(* IEC 61131-3 sources: com.logicals.lc3.webinar/usRTS_RPMControl_iSOC/src_FB_LIB_SAFE/Convert/ULINT, 4 files *)

(* ---- wTRUNC_ULINT_TO_UDINT.iecst ---- *)
NAMESPACE logicals.web.standard
NAMESPACE convert

/*
 * Function block wrapper for IEC 61131-3 TO_UDINT<br>
 * IN =  input value (ULINT)<br>
 * OUT = IN (UDINT)<br>
 */
FUNCTION_BLOCK wTRUNC_ULINT_TO_UDINT
	{ vNameAlignment:="center"; altName:="TRUNC_ULINT_TO_UDINT"; bgColor:="Plum"; width:=180; hideIONames; }
	VAR_INPUT
		IN : ULINT;
	END_VAR
	VAR_OUTPUT
		OUT: UDINT;
	END_VAR

	OUT := TO_UDINT(IN:=IN, ENO=>ENO);
END_FUNCTION_BLOCK

END_NAMESPACE
END_NAMESPACE

(* ---- wTRUNC_ULINT_TO_UINT.iecst ---- *)
NAMESPACE logicals.web.standard
NAMESPACE convert

/*
 * Function block wrapper for IEC 61131-3 TO_UINT<br>
 * IN =  input value (ULINT)<br>
 * OUT = IN (UINT)<br>
 */
FUNCTION_BLOCK wTRUNC_ULINT_TO_UINT
	{ vNameAlignment:="center"; altName:="TRUNC_ULINT_TO_UINT"; bgColor:="Plum"; width:=180; hideIONames; }
	VAR_INPUT
		IN : ULINT;
	END_VAR
	VAR_OUTPUT
		OUT: UINT;
	END_VAR

	OUT := TO_UINT(IN:=IN, ENO=>ENO);
END_FUNCTION_BLOCK

END_NAMESPACE
END_NAMESPACE

(* ---- wTRUNC_ULINT_TO_USINT.iecst ---- *)
NAMESPACE logicals.web.standard
NAMESPACE convert

/*
 * Function block wrapper for IEC 61131-3 TO_USINT<br>
 * IN =  input value (ULINT)<br>
 * OUT = IN (USINT)<br>
 */
FUNCTION_BLOCK wTRUNC_ULINT_TO_USINT
	{ vNameAlignment:="center"; altName:="TRUNC_ULINT_TO_USINT"; bgColor:="Plum"; width:=180; hideIONames; }
	VAR_INPUT
		IN : ULINT;
	END_VAR
	VAR_OUTPUT
		OUT: USINT;
	END_VAR

	OUT := TO_USINT(IN:=IN, ENO=>ENO);
END_FUNCTION_BLOCK

END_NAMESPACE
END_NAMESPACE

(* ---- wULINT_TO_LWORD.iecst ---- *)
NAMESPACE logicals.web.standard
NAMESPACE convert

/*
 * Function block wrapper for IEC 61131-3 TO_LWORD<br>
 * IN =  input value (ULINT)<br>
 * OUT = IN (LWORD)<br>
 */
FUNCTION_BLOCK wULINT_TO_LWORD
	{ vNameAlignment:="center"; altName:="ULINT_TO_LWORD"; bgColor:="DodgerBlue"; width:=140; hideIONames; }
	VAR_INPUT
		IN : ULINT;
	END_VAR
	VAR_OUTPUT
		OUT: LWORD;
	END_VAR

	OUT := TO_LWORD(IN:=IN, ENO=>ENO);
END_FUNCTION_BLOCK

END_NAMESPACE
END_NAMESPACE
